Staubli VAL3: test.dtx

mdesc mNomSpeed
string sTarget{}
  [Key1] = {}
string sOrig{}
  [Key1] = {}
  [Key2] = {}
  [Key3] = {}
  [Key4] = {}
  [Key5] = {}
  [Key6] = {}
  [Key7] = {}
  [Key8] = {}
  [Key9] = {}
  [Key10] = {}
string sKey
